FUNCTION_BLOCK FB_FSM_Diagnostic
VAR_INPUT
	stIn : ST_FSM_In;
	stOut : ST_FSM_Out;
	stParams : ST_FSM_Params;
	stCtrl : ST_FSM_Ctrl;
	bHwError : BOOL;
	bAck : BOOL;
	stStatus : ST_FSM_Status;	
END_VAR
VAR_IN_OUT
END_VAR
VAR_OUTPUT
	bCritical	: BOOL;
	bError		: BOOL;
	bWarning	: BOOL;
	bInfo		: BOOL;
	bVerbose	: BOOL;
	bFailure	: BOOL;
	bBlinking	: BOOL;
	bFixed		: BOOL;
END_VAR
VAR
END_VAR

// on Ack, reset holding conditions
IF bAck THEN
	bCritical := FALSE;
	bError := FALSE;
	bWarning := FALSE;
	bInfo := FALSE;
	bVerbose := FALSE;
	bBlinking := FALSE;
END_IF

// update critical condition

// update holding conditions
bFailure := bCritical OR bError;

bBlinking := bFailure;
bFixed := bWarning;

END_FUNCTION_BLOCK

(* stored: Version 1.1.0.1
   POU FB_FSM_Diagnostic: Id {c0576ddd-8680-01ec-1943-b48faece56d8}, SpecialFunc None *)
